(* IEC 61131-3 sources: repolevel_ST_code_completion/output/0121完整版本/repoeval_electronic_gear_motion/readful_result_no_provide, 2 files *)

(* ---- FB_DualAxisPower.st ---- *)
VAR
	fbPower1		:	MC_Power;		//轴1电源控制
	fbPower2		:	MC_Power;		//轴2电源控制
	bAxis1Error		:	BOOL;			//轴1错误标志
	bAxis2Error		:	BOOL;			//轴2错误标志
END_VAR

fbPower1(
	Axis := Axis1,
	Enable := bEnable,
	bDriveStart := TRUE,
	bRegulatorOn := TRUE
);

fbPower2(
	Axis := Axis2,
	Enable := bEnable,
	bDriveStart := TRUE,
	bRegulatorOn := TRUE
);

bAxis1Ready := fbPower1.Status = MC_POWER_STATUS_READY;
bAxis2Ready := fbPower2.Status = MC_POWER_STATUS_READY;

bAxis1Error := fbPower1.Error;
bAxis2Error := fbPower2.Error;

bError := bAxis1Error OR bAxis2Error;

bBothReady := bAxis1Ready AND bAxis2Ready;
END_FUNCTION_BLOCK

(* ---- FB_GearMotionControl.st ---- *)
VAR
	fbPowerMgr			:	FB_DualAxisPower;	//双轴电源管理
	fbGearCtrl			:	FB_GearCoupling;	//齿轮耦合控制
	fbMoveVel			:	MC_MoveVelocity;	//速度运动
	fbHaltMaster		:	MC_Halt;			//主轴停止
	fbHaltSlave			:	MC_Halt;			//从轴停止
	fbStartRtrig		:	R_TRIG;				//启动上升沿
	fbStopRtrig			:	R_TRIG;				//停止上升沿
	nState				:	BYTE;				//内部状态机
	bMasterReady		:	BOOL;				//主轴准备就绪
	bSlaveReady			:	BOOL;				//从轴准备就绪
END_VAR

fbStartRtrig(CLK := bStart);
fbStopRtrig(CLK := bStop);

CASE nState OF
	0: (* 等待轴准备就绪 *)
		fbPowerMgr(
			Axis1 := MasterAxis,
			Axis2 := SlaveAxis,
			bEnable := TRUE
		);
		bMasterReady := fbPowerMgr.bAxis1Ready;
		bSlaveReady := fbPowerMgr.bAxis2Ready;

		IF bMasterReady AND bSlaveReady THEN
			bReady := TRUE;
			nState := 1;
		END_IF;

	1: (* 启动运动 *)
		IF fbStartRtrig.Q THEN
			fbMoveVel(
				Axis := MasterAxis,
				Velocity := rVelocity,
				Acceleration := rAcceleration,
				Deceleration := rDeceleration,
				Direction := nDirection,
				Execute := TRUE
			);
			IF fbMoveVel.Done THEN
				fbGearCtrl(
					Master := MasterAxis,
					Slave := SlaveAxis,
					RatioNumerator := nRatioNumerator,
					RatioDenominator := nRatioDenominator,
					Execute := TRUE
				);
				IF fbGearCtrl.Done THEN
					bRunning := TRUE;
					nState := 2;
				END_IF;
			END_IF;
		END_IF;

	2: (* 运行中 *)
		IF fbStopRtrig.Q THEN
			fbHaltMaster(
				Axis := MasterAxis,
				Execute := TRUE
			);
			fbHaltSlave(
				Axis := SlaveAxis,
				Execute := TRUE
			);
			IF fbHaltMaster.Done AND fbHaltSlave.Done THEN
				bRunning := FALSE;
				nState := 0;
			END_IF;
		END_IF;

	ELSE
		bError := TRUE;
END_CASE;

nCurrentState := nState;
END_FUNCTION_BLOCK
